// TIA Portal V19 export
TYPE "LEXCHANGETRAY_typeHandlingXyzIoSignalInterface"
// configuration: LEXCHANGETRAY_typeHandlingXyzIoSignalConfigeration
// commands: LEXCHANGETRAY_typeHandlingXyzIoSignalManualCommands
// monitoring: LEXCHANGETRAY_typeHandlingXyzIoSignalProcessValues
// stored: Access Published
   STRUCT
      configuration : "LEXCHANGETRAY_typeHandlingXyzIoSignalConfigeration";
      commands { S7_SetPoint := 'True'} : "LEXCHANGETRAY_typeHandlingXyzIoSignalManualCommands";
      monitoring { S7_SetPoint := 'True'} : "LEXCHANGETRAY_typeHandlingXyzIoSignalProcessValues";
   END_STRUCT;
END_TYPE
